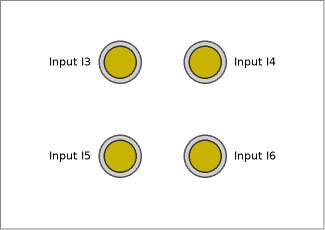
VISUALIZATION V_DI  // 325x230
    Lamp1 (95,37 50x50), variable: Module_IO.iTestInput[3], style: Lamp-Lamp1-Yellow
    Lamp1 (180,37 50x50), variable: Module_IO.iTestInput[4], style: Lamp-Lamp1-Yellow
    Lamp1 (95,131 50x50), variable: Module_IO.iTestInput[5], style: Lamp-Lamp1-Yellow
    Lamp1 (180,131 50x50), variable: Module_IO.iTestInput[6], style: Lamp-Lamp1-Yellow
    Label (40,47 60x30), "Input I3"
    Label (40,141 60x30), "Input I5"
    Label (225,47 60x30), "Input I4"
    Label (225,141 60x30), "Input I6"
END_VISUALIZATION

(* stored: Version 1.1.0.1, ProductVersion 3.1.4024.11
   Visu V_DI: Id {61e375e9-302e-40be-8686-5bebaf65ba78} *)
